FUNCTION "FC_Crt_ICSExcepTrac" : VOID
TITLE =%version: 0.02 % CN: 32
//Function:
//Prepare and send message 'ICS Exception Trace' - TIR record
//
//History:
//This version  %created_by: nlhdl %
//              %date_created: Thursday, November 02, 2017 9:04:01 AM %
//              %release: VI_GEN/RA_Dev %
//
//Modification History:                                 By:      Date:     Rev:
//----------------------------------------------------  -------  --------  -----
//ra#26038: ICSExceptionTrace use TIC                   nlHdL    02-11-17   0.02
//Initial Version                                       nlHdL    17-02-17   0.01
//
//Description:
//Prepare and send message 'ICS Exception' - Tubtrace function
//
FAMILY : VIBES
VERSION : 0.0


VAR_INPUT
  i_ID : DWORD ;	//ID Record HEX AAAA - ZZSS/OO.
  i_DB_Event_Num : INT ;	//Number of DB event
  i_FIFO_PLC_DB_num : INT ;	//Number of DB PLC FIFO
  i_Event_value : INT ;	//Event Value IILLL = II = ICS Event number LLL = LNK number
END_VAR
VAR_TEMP
  t_AR1_Backup : DINT ;	//Save the contents of AR1
  t_Ret_Val_Word : WORD ;	//Return value
  t_Ret_Val_Int : INT ;	//Return Value
  t_Text_Clear_Counter : INT ;	//Counter to clear all text characters
  t_Next_Adress : INT ;	//Next adress to clear
  t_Start_Adress : INT ;	//Start adress in DB_outgoing_Msgs of Logging Messages
  t_LNK : INT ;	//LNK Number
  t_TIC : INT ;	//TIC Number
END_VAR
BEGIN
NETWORK
TITLE =AA: Store AR1 and Get Date and Time

      TAR1  ; // Store AR1
      T     #t_AR1_Backup;

      CALL "READ_CLK" (
           RET_VAL                  := #t_Ret_Val_Int,
           CDT                      := "DB_Outgoing_Msgs".ICSExceptionTrace.EventTime);

NETWORK
TITLE =BA: Write messageID

      L     2603;
      T     "DB_Outgoing_Msgs".ICSExceptionTrace.MessageID;
NETWORK
TITLE =CA: Copy AreaID, ZoneID and SectionID

      L     #i_ID; // Load ID
      L     DW#16#FFFF0000; // Filter Area number only
      AD    ;
      SRD   16; // Slide Area nubmer to beginning AAAA0000 -> AAAA
      BTD   ; // Convert HEX to INT
      T     "DB_Outgoing_Msgs".ICSExceptionTrace.AreaID; // Transfer to outgoing messages

      L     #i_ID; // Load ID
      L     DW#16#FF00; // Filter Zone number only
      AD    ;
      SRD   8; // Slide Zone nubmer to beginning 0000ZZ00 -> 0000ZZ
      BTI   ; // Convert HEX to INT
      T     "DB_Outgoing_Msgs".ICSExceptionTrace.ZoneID; // Transfer to outgoing messages

      L     #i_ID; // Load ID
      L     DW#16#FF; // Filter Section number only
      AD    ;
      BTI   ; // Convert HEX to INT
      T     "DB_Outgoing_Msgs".ICSExceptionTrace.EquipmentID; // Transfer to outgoing messages
NETWORK
TITLE =DA: Write data to log messages

      L     #i_Event_value;
      L     1000;
      /D    ;
      T     "DB_Outgoing_Msgs".ICSExceptionTrace.ICSEvent; // Transfer to outgoing messages
      L     1000;
      *I    ;
      T     #t_Ret_Val_Int;
      L     #i_Event_value;
      L     #t_Ret_Val_Int;
      -I    ;
      T     #t_LNK;

      CALL "FC_Read_Int_Record" (
           i_Record_Number          := #t_LNK,
           i_P_INT_Record           := "DB_UDT_LNK_Record".TIC,
           i_DB                     := "DB_LNK_List",
           i_DB_Event_Num           := #i_DB_Event_Num,
           o_INT                    := #t_TIC);

      L     #t_TIC;
      T     "DB_Outgoing_Msgs".ICSExceptionTrace.TIC;

      CALL "FC_Read_ANY_Record" (
           i_Record_Number          := #t_TIC,
           i_ANY_Data_Record        := "DB_UDT_TIC_Record".TIR,
           i_ANY_Data               := "DB_Outgoing_Msgs".ICSExceptionTrace.Carrier,
           i_DB                     := "DB_TIC_List",
           i_DB_Event_Num           := #i_DB_Event_Num);

NETWORK
TITLE =EA: Put message in buffer

      CALL "BLKMOV" (
           SRCBLK                   := "DB_Outgoing_Msgs".Default,
           RET_VAL                  := #t_Ret_Val_Int,
           DSTBLK                   := "DB_Outgoing_Msgs".Merged_Message);

      CALL "BLKMOV" (
           SRCBLK                   := "DB_Outgoing_Msgs".ICSExceptionTrace,
           RET_VAL                  := #t_Ret_Val_Int,
           DSTBLK                   := "DB_Outgoing_Msgs".Merged_Message);

      CALL "FC_FIFO" (
           i_FIFO_DB_Num            := #i_FIFO_PLC_DB_num,
           i_Mode                   := 'L',
           i_ANY_Data               := "DB_Outgoing_Msgs".Merged_Message,
           i_ID                     := #i_ID,
           o_RET_VAL_FIFO           := #t_Ret_Val_Word);

NETWORK
TITLE =FA: Clear Text with spaces
//Clear text after the message to be enable to add the detailed text to the
//message.
//Clear the text for new messages within text.
      OPN   "DB_Outgoing_Msgs";
      L     0;
      T     #t_Text_Clear_Counter;

      CALL "FC_Any_To_Adress" (
           i_ANY_Data               := "DB_Outgoing_Msgs".ICSExceptionTrace.ICSEventDetail,
           o_Adress                 := #t_Start_Adress);

FA01: L     #t_Start_Adress;
      L     #t_Text_Clear_Counter;
      +I    ;
      T     #t_Next_Adress;
      SLW   3;
      LAR1  ;

      L     ' ';
      T     DBB [AR1,P#0.0];

      L     #t_Text_Clear_Counter;
      L     1;
      +I    ;
      T     #t_Text_Clear_Counter;
      L     100;
      >=I   ;
      JCN   FA01;

      L     #t_Next_Adress;
NETWORK
TITLE =GA: Restore AR1

      L     #t_AR1_Backup;
      LAR1  ;
END_FUNCTION

